{attribute 'Tc2GvlVarNames'}
{attribute 'strict'}
// Stato del Punto di Prelievo 
TYPE e_Stato_PickPoint :
(
	WORKPICKPOINT_STATE_MAN			:= 0,	(* PickPoint in Stato Manuale *)
	WORKPICKPOINT_STATE_AUTO		:= 1,	(* PickPoint in Stato Automatico *)	
	WORKPICKPOINT_STATE_ERROR		:= 99 (* PickPoint in Stato di Errore *)
);
END_TYPE

(* stored: Version 1.1.0.1, ProductVersion 3.1.4024.11
   EnumerationTextList e_Stato_PickPoint: Id {92f19b3d-bdf3-4428-a075-f8e1cba6c143} *)
